// TIA Portal project "Product_Automation_Project" (V17)

(* hardware
DEVICE "S7-1200 station_1"  S7-1200 Station
   slot 0: "Rack_0"  S7-1200 Rack  Rack  V1.0
   slot 1: "PLC_1"  CPU 1214C AC/DC/Rly  6ES7 214-1BG40-0XB0  V4.5
   slot 3: "AQ 1x12BIT_1"  AQ1 signal board  6ES7 232-4HA30-0XB0  V1.0
*)

// ===== PLC "PLC_1"  CPU 1214C AC/DC/Rly =====

VAR_GLOBAL   // PLC tag table "Inputs"
   "PI-100" AT %IW64 : Int;   // Pressure tank sensor
   "H-100.1" AT %I0.1 : Bool;   // System start button
   "H-100.2" AT %I0.2 : Bool;   // System stop button
   "H-100.3" AT %I0.4 : Bool;   // Emergency stop button
   "H-100.4" AT %I0.5 : Bool;   // Emergency reset
   "H-100.5" AT %I0.6 : Bool;   // Pressure tank emptying button
   "Brush_state" AT %I0.0 : Bool;
   "H-100.6" AT %I0.7 : Bool;   // Maintenance reset
END_VAR

VAR_GLOBAL   // PLC tag table "Outputs"
   "PC-100" AT %QW64 : Int;   // Air compressor control
   "OI-100.1" AT %Q0.1 : Bool;   // PID on
   "OI-100.2" AT %Q0.2 : Bool;   // PID off
   "OI-100.3" AT %Q0.3 : Bool;   // Led pressure alarm
   "OI-100.4" AT %Q0.4 : Bool;   // Emergency valve open
   "OI-100.5" AT %Q0.5 : Bool;   // Brush valve closed
   "OI-100.6" AT %Q0.6 : Bool;   // Empty tank indicator
   "OI-100.7" AT %Q0.7 : Bool;
END_VAR

VAR_GLOBAL   // PLC tag table "Variables"
   "PI-100.n" AT %MD0 : Real;   // normalized PI-100 value
   "PI-100.r" AT %MD6 : Real;   // real PI-100 value
   "PC-100.r" AT %MD1 : Real;   // real PC-100 value
   "PC-100.n" AT %MD8 : Real;   // normalized PC-100 value
   "PI-100.r2" AT %MD12 : Real;   // tank pressure
   "System_output" AT %MD16 : Real;   // true system output
   "Brush_pressure" AT %MD20 : Real;   // The ouput pressure of the brush
   "Flip-Flop" AT %M24.0 : Bool;   // Flip-flop
   "Start/Stop value" AT %M24.1 : Bool;
   "Emergency value" AT %M24.2 : Bool;
   "System_state" AT %M24.3 : Bool;
   "Max_pressure_reached" AT %M24.4 : Bool;
   "Emergency_pressure" AT %MD34 : Real;
   "Maintenance_state" AT %M24.5 : Bool;
   "Maintenance_pressure" AT %MD28 : Real;
   "Flip-Flop(1)" AT %M32.0 : Bool;
   "Flip-Flop(2)" AT %M32.1 : Bool;
   "Reset value" AT %M32.2 : Bool;
   "Pressure alarm" AT %M32.4 : Bool;
   "Emergency state" AT %M32.5 : Bool;
   "Brush active/inactive" AT %M32.6 : Bool;
   "min_Output_Reached" AT %M32.7 : Bool;
END_VAR

VAR_GLOBAL   // PLC tag table "Clock_pulses"
   "Clock_Byte(1)" AT %MB150 : Byte;
   "Clock_10Hz(1)" AT %M150.0 : Bool;
   "Clock_5Hz(1)" AT %M150.1 : Bool;
   "Clock_2.5Hz(1)" AT %M150.2 : Bool;
   "Clock_2Hz(1)" AT %M150.3 : Bool;
   "Clock_1.25Hz(1)" AT %M150.4 : Bool;
   "Clock_1Hz(1)" AT %M150.5 : Bool;
   "Clock_0.625Hz(1)" AT %M150.6 : Bool;
   "Clock_0.5Hz(1)" AT %M150.7 : Bool;
END_VAR

DATA_BLOCK "Bool->Real_DB"   // DB1
{ S7_Optimized_Access := 'TRUE' }
VERSION : 0.1
// stored: InstanceOfName Bool->Real
"Bool->Real"
BEGIN
END_DATA_BLOCK

DATA_BLOCK "Integrating_process_DB"   // DB4
{ S7_Optimized_Access := 'TRUE' }
VERSION : 2.01
// stored: InstanceOfName LSim_I
"LSim_I"
BEGIN
END_DATA_BLOCK

DATA_BLOCK "System_state_FB_DB"   // DB5
{ S7_Optimized_Access := 'TRUE' }
VERSION : 0.1
// stored: InstanceOfName System_state_FB
"System_state_FB"
BEGIN
END_DATA_BLOCK

DATA_BLOCK "Emergency_valve_open_DB"   // DB6
{ S7_Optimized_Access := 'TRUE' }
VERSION : 0.1
// stored: InstanceOfName Bool->Real
"Bool->Real"
BEGIN
END_DATA_BLOCK

DATA_BLOCK "Maintenance_DB"   // DB7
{ S7_Optimized_Access := 'TRUE' }
VERSION : 0.1
// stored: InstanceOfName Bool->Real
"Bool->Real"
BEGIN
END_DATA_BLOCK

DATA_BLOCK "Leds_Logic_DB"   // DB8
{ S7_Optimized_Access := 'TRUE' }
VERSION : 0.1
// stored: InstanceOfName Leds_Logic
"Leds_Logic"
BEGIN
END_DATA_BLOCK

DATA_BLOCK "Pressure_alarm_DB"   // DB10
{ S7_Optimized_Access := 'TRUE' }
VERSION : 0.1
// stored: InstanceOfName Pressure_alarm
"Pressure_alarm"
BEGIN
END_DATA_BLOCK

FUNCTION_BLOCK "Signal_scaling"   // FB1, LAD
TITLE = Signal scaling
{ S7_Optimized_Access := 'TRUE' }
VERSION : 0.1
// Here we have the process of scaling the input signal of the PID
   VAR_INPUT
      Input_value : Int;
   END_VAR
   VAR_OUTPUT
      Output_value : Real;
   END_VAR
   VAR_IN_OUT
      Normalized_value : Real;
   END_VAR
BEGIN

REGION Network 1: Normalizing input value
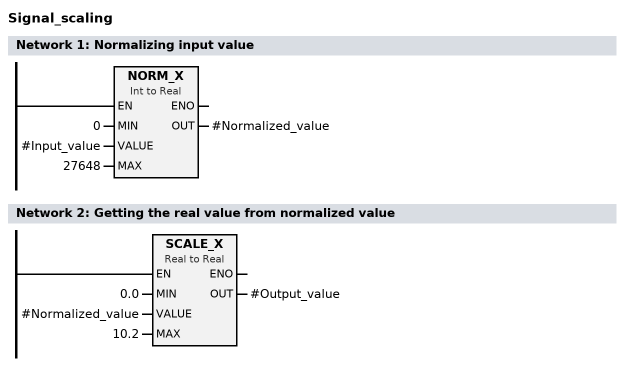
   RUNG wire#powerrail
      { S7_Templates := "[SrcType := Int, DestType := Real]" } Normalize(min := 0, value := #Input_value, max := 27648, out => #Normalized_value)
   END_RUNG
   // the same network as SCL:
   #Normalized_value := NORM_X(MIN := 0, VALUE := #Input_value, MAX := 27648);
END_REGION

REGION Network 2: Getting the real value from normalized value
   RUNG wire#powerrail
      { S7_Templates := "[SrcType := Real, DestType := Real]" } Scale(min := 0.0, value := #Normalized_value, max := 10.2, out => #Output_value)
   END_RUNG
   // the same network as SCL:
   #Output_value := SCALE_X(MIN := 0.0, VALUE := #Normalized_value, MAX := 10.2);
END_REGION
END_FUNCTION_BLOCK

FUNCTION_BLOCK "Bool->Real"   // FB2, SCL
{ S7_Optimized_Access := 'TRUE' }
VERSION : 0.1
   VAR_INPUT
      Boolean_input : Bool;
      Input_pressure : Real;
   END_VAR
   VAR_OUTPUT
      Output_pressure : Real;
   END_VAR
BEGIN
   IF #Boolean_input THEN
       #Output_pressure := #Input_pressure;
   ELSE
       #Output_pressure := 0;
   END_IF;
END_FUNCTION_BLOCK

FUNCTION_BLOCK "System_state_FB"   // FB3, FBD
TITLE = System functioning logic
{ S7_Optimized_Access := 'TRUE' }
VERSION : 0.1
BEGIN

REGION Network 1: System state logic
   // Both Emergency value and Start/Stop value must be "1"
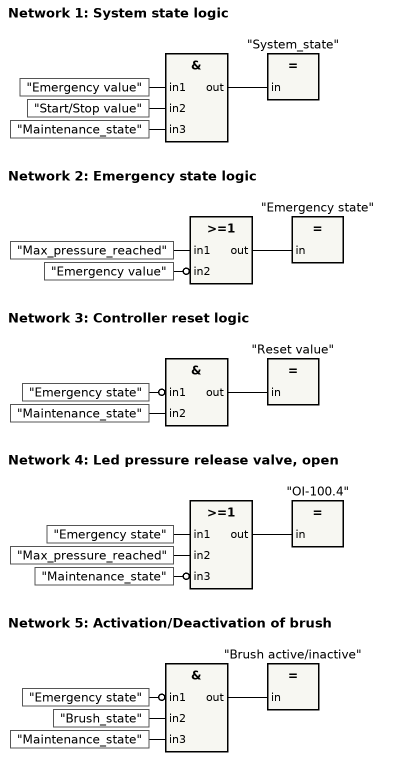
   "System_state" := "Emergency value" AND "Start/Stop value" AND "Maintenance_state";
END_REGION

REGION Network 2: Emergency state logic
   // if max pressure (10.5) is reached or emergency value is 1 than the emergency state is "1"
   "Emergency state" := "Max_pressure_reached" OR NOT "Emergency value";
END_REGION

REGION Network 3: Controller reset logic
   // If both are not pressed then Reset value is 1 -> 0 in controller
   "Reset value" := NOT "Emergency state" AND "Maintenance_state";
END_REGION

REGION Network 4: Led pressure release valve, open
   "OI-100.4" := "Emergency state" OR "Max_pressure_reached" OR NOT "Maintenance_state";
END_REGION

REGION Network 5: Activation/Deactivation of brush
   // Emergency state is active when 0 and inactive when 1
   "Brush active/inactive" := NOT "Emergency state" AND "Brush_state" AND "Maintenance_state";
END_REGION
END_FUNCTION_BLOCK

FUNCTION_BLOCK "Leds_Logic"   // FB4, SCL
{ S7_Optimized_Access := 'TRUE' }
VERSION : 0.1
   VAR_INPUT
      Input : Bool;
   END_VAR
   VAR_OUTPUT
      Output1 : Bool;
      Output2 : Bool;
   END_VAR
BEGIN
   IF #Input THEN
       #Output1 := 1;
       #Output2 := 0;
   ELSE
       #Output2 := 1;
       #Output1 := 0;
   END_IF;
END_FUNCTION_BLOCK

FUNCTION_BLOCK "Pressure_alarm"   // FB5, SCL
{ S7_Optimized_Access := 'TRUE' }
VERSION : 0.1
   VAR_INPUT
      Input : Real;
   END_VAR
   VAR_OUTPUT
      Output : Bool;
   END_VAR
BEGIN
   IF #Input>=10.2 AND #Input<10.5 THEN
       #Output := 1;
   ELSE
       #Output := 0;
   END_IF;
END_FUNCTION_BLOCK

FUNCTION_BLOCK "LSim_I"   // FB56, SCL
{ S7_Optimized_Access := 'TRUE' }
VERSION : 2.01
   VAR_INPUT
      calcParam : Bool;   // recalculate with new parameters
      input : Real;   // input signal
      tmLag1 : Real := 1.0;   // time constant T1 [sec]
      cycle : Real := 0.1;   // cyclic time [sec]
      maxOut : Real := 100.0;   // max. output limit
      minOut : Real;   // min. output limit
      reset : Bool;   // resets all relevant parameters to ‘0’ including the output
   END_VAR
   VAR_OUTPUT
      error : Bool;   // error (#tmLag1 <= 0)
      status : Word;   // status (if #tmLag1 <= 0 then status = 16#8001)
      maxReached : Bool;   // output has reached max. limit
      minReached : Bool;   // output has reached min. limit
      output : Real;   // output signal (if #error = FALSE)
   END_VAR
   VAR
      statRxn1 : Real;   // delayed input signal (n-1)
      statRyn1 : Real;   // delayed output signal (n-1)
      statRa1 : Real;
      statRb1 : Real;
      statOverfirst : Bool;
      statOutput : Real;   // output signal
   END_VAR
BEGIN
   //=============================================================================
   //SIEMENS AG
   //(c)Copyright 2017 All Rights Reserved
   //-----------------------------------------------------------------------------
   //Library:       Library for Controlled System Simulation
   //Tested with:   S7-1500 FW V2.0 / S7-1200 FW V4.2
   //Engineering:   STEP 7 V14 Upd2 (TIA Portal)
   //Restrictions:  Cyclic interrupt
   //Requirements:  memory card needed for S7-1500
   //Functionality: Simulation of a I-System
   //
   //             1
   //  F(p) = -----------
   //         (tmLag1*p)
   //          
   //  Call the simulation in a cyclic interrupt with
   //  cyclic interrupt time at least = tmLag1/10!
   //-----------------------------------------------------------------------------
   //Change log table:
   //Version  Date       Expert in charge                Changes applied
   //02.00.00 03.02.2016 Siemens Industry Online Support Release (STEP 7 V13 SP1)
   //02.00.01 02.03.2017 Siemens Industry Online Support Release (STEP 7 V14)
   //=============================================================================

   // check parameter
   IF #tmLag1 <= 0 THEN
     #error := True;
     #status := W#16#8001;     // Parameter Error
     #statRxn1 := 0.0;
     #statRyn1 := 0.0;
     #statOutput := 0;
     #output := 0;
     RETURN;
   ELSE
     #error := FALSE;
     #status := W#16#0000;     // no error
   END_IF;

   // calculates the z-parameter for the difference equatation
   IF #calcParam = True OR NOT #statOverfirst THEN
   #statOverfirst:=1;
     // Calculate z-parameters for IT1-System
   #statRb1 := #cycle/#tmLag1;
   #statRa1 := -1;

   END_IF;

   // reset Memory
   IF #reset = True THEN
     #statRxn1 := 0.0;
     #statRyn1 := 0.0;
     #statOutput:=0;
   END_IF;

   // save delayed output-signals
   #statRyn1:= #statOutput;

   // difference equatation for the I-system
   #statOutput := #statRxn1* #statRb1 - #statRyn1*#statRa1;

   // save delayed input-signals
   #statRxn1 := #input;

   // max limit of acutating variable
   IF #statOutput > #maxOut THEN
     #statOutput := #maxOut;
     #maxReached:= True;
   ELSE
     #maxReached := False;
   END_IF;

   // min limit of acutating variable
   IF #statOutput < #minOut THEN
     #statOutput := #minOut;
     #minReached := True;
   ELSE
     #minReached := False;
   END_IF;

   #output := #statOutput;
END_FUNCTION_BLOCK

ORGANIZATION_BLOCK "Main"   // OB1, LAD, ProgramCycle
TITLE = "Main Program Sweep (Cycle)"
{ S7_Optimized_Access := 'TRUE' }
VERSION : 0.1
   VAR_INPUT
      Initial_Call : Bool;   // Initial call of this OB
      Remanence : Bool;   // =True, if remanent data are available
   END_VAR
BEGIN

REGION Network 1: Start/Stop logic
   // if start button is pressed then Start/Stop value becomes 1 and if emergency value is also 1 then system state is 1
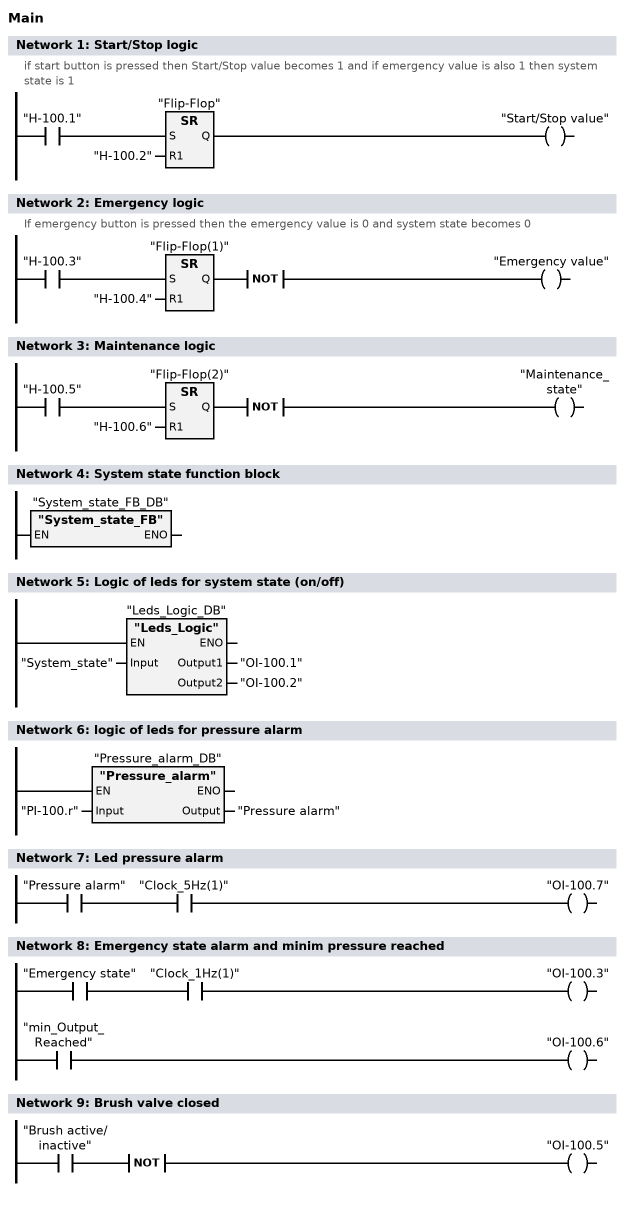
   RUNG wire#powerrail
      Contact( "H-100.1" )
      S_SR(operand := "Flip-Flop", r1 := "H-100.2")
      Coil( "Start/Stop value" )
   END_RUNG
   // the same network as SCL:
   IF "H-100.1" THEN
       "Flip-Flop" := TRUE;   // SR flip-flop
   END_IF;
   IF "H-100.2" THEN "Flip-Flop" := FALSE; END_IF;
   "Start/Stop value" := "Flip-Flop";
END_REGION

REGION Network 2: Emergency logic
   // If emergency button is pressed then the emergency value is 0 and system state becomes 0
   RUNG wire#powerrail
      Contact( "H-100.3" )
      S_SR(operand := "Flip-Flop(1)", r1 := "H-100.4")
      Not()
      Coil( "Emergency value" )
   END_RUNG
   // the same network as SCL:
   IF "H-100.3" THEN
       "Flip-Flop(1)" := TRUE;   // SR flip-flop
   END_IF;
   IF "H-100.4" THEN "Flip-Flop(1)" := FALSE; END_IF;
   "Emergency value" := NOT "Flip-Flop(1)";
END_REGION

REGION Network 3: Maintenance logic
   RUNG wire#powerrail
      Contact( "H-100.5" )
      S_SR(operand := "Flip-Flop(2)", r1 := "H-100.6")
      Not()
      Coil( "Maintenance_state" )
   END_RUNG
   // the same network as SCL:
   IF "H-100.5" THEN
       "Flip-Flop(2)" := TRUE;   // SR flip-flop
   END_IF;
   IF "H-100.6" THEN "Flip-Flop(2)" := FALSE; END_IF;
   "Maintenance_state" := NOT "Flip-Flop(2)";
END_REGION

REGION Network 4: System state function block
   RUNG wire#powerrail
      "System_state_FB_DB"()
   END_RUNG
   // the same network as SCL:
   "System_state_FB_DB"();   // "System_state_FB"
END_REGION

REGION Network 5: Logic of leds for system state (on/off)
   RUNG wire#powerrail
      "Leds_Logic_DB"(Input := "System_state", Output1 => "OI-100.1", Output2 => "OI-100.2")
   END_RUNG
   // the same network as SCL:
   "Leds_Logic_DB"(Input := "System_state", Output1 => "OI-100.1", Output2 => "OI-100.2");   // "Leds_Logic"
END_REGION

REGION Network 6: logic of leds for pressure alarm
   RUNG wire#powerrail
      "Pressure_alarm_DB"(Input := "PI-100.r", Output => "Pressure alarm")
   END_RUNG
   // the same network as SCL:
   "Pressure_alarm_DB"(Input := "PI-100.r", Output => "Pressure alarm");   // "Pressure_alarm"
END_REGION

REGION Network 7: Led pressure alarm
   RUNG wire#powerrail
      Contact( "Pressure alarm" )
      Contact( "Clock_5Hz(1)" )
      Coil( "OI-100.7" )
   END_RUNG
   // the same network as SCL:
   "OI-100.7" := "Pressure alarm" AND "Clock_5Hz(1)";
END_REGION

REGION Network 8: Emergency state alarm and minim pressure reached
   RUNG wire#powerrail
      Contact( "Emergency state" )
      Contact( "Clock_1Hz(1)" )
      Coil( "OI-100.3" )
   END_RUNG
   RUNG wire#powerrail
      Contact( "min_Output_Reached" )
      Coil( "OI-100.6" )
   END_RUNG
   // the same network as SCL:
   "OI-100.3" := "Emergency state" AND "Clock_1Hz(1)";
   "OI-100.6" := "min_Output_Reached";
END_REGION

REGION Network 9: Brush valve closed
   RUNG wire#powerrail
      Contact( "Brush active/inactive" )
      Not()
      Coil( "OI-100.5" )
   END_RUNG
   // the same network as SCL:
   "OI-100.5" := NOT "Brush active/inactive";
END_REGION
END_ORGANIZATION_BLOCK

ORGANIZATION_BLOCK "Cyclic interrupt_1"   // OB30, FBD, CyclicInterrupt
TITLE = Main control loop
{ S7_Optimized_Access := 'TRUE' }
VERSION : 0.1
   VAR_INPUT
      Initial_Call : Bool;   // Initial call of this OB
      Event_Count : Int;   // Events discarded
   END_VAR
BEGIN

REGION Network 1: PID
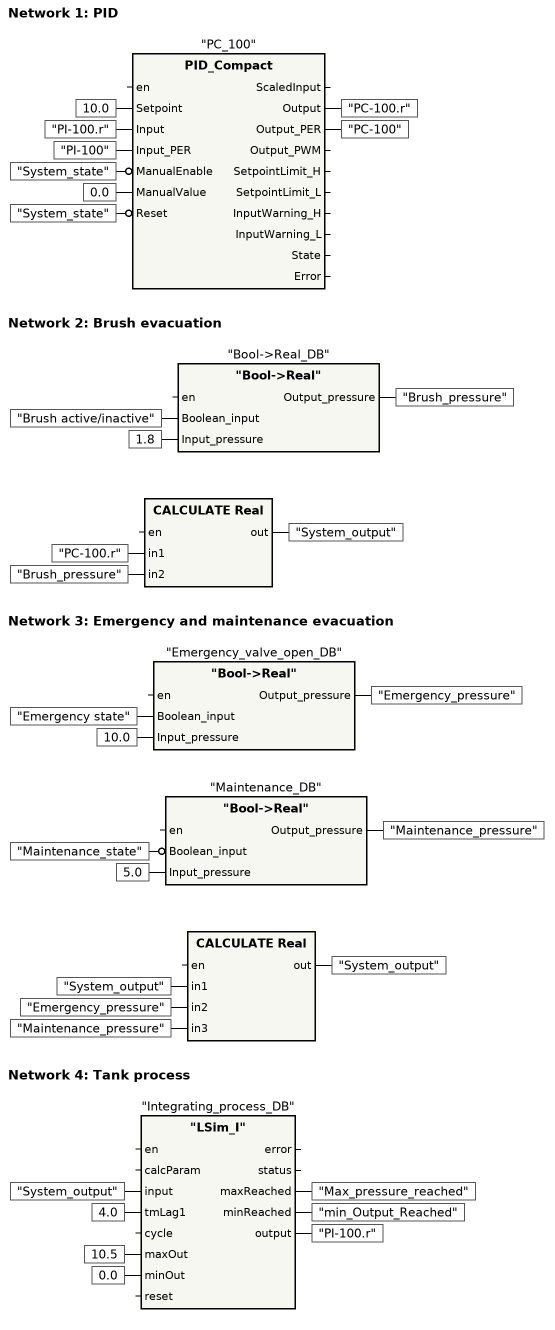
   "PC_100"(Setpoint := 10.0,   // PID_Compact
            Input := "PI-100.r",
            Input_PER := "PI-100",
            ManualEnable := NOT "System_state",
            ManualValue := 0.0,
            Reset := NOT "System_state",
            Output => "PC-100.r",
            Output_PER => "PC-100");
END_REGION

REGION Network 2: Brush evacuation
   "Bool->Real_DB"(Boolean_input := "Brush active/inactive",   // "Bool->Real"
                   Input_pressure := 1.8,
                   Output_pressure => "Brush_pressure");
   "System_output" := "PC-100.r"-"Brush_pressure";
END_REGION

REGION Network 3: Emergency and maintenance evacuation
   "Emergency_valve_open_DB"(Boolean_input := "Emergency state",   // "Bool->Real"
                           Input_pressure := 10.0,
                           Output_pressure => "Emergency_pressure");
   "Maintenance_DB"(Boolean_input := NOT "Maintenance_state",   // "Bool->Real"
                    Input_pressure := 5.0,
                    Output_pressure => "Maintenance_pressure");
   "System_output" := "System_output"- "Emergency_pressure" - "Maintenance_pressure";
END_REGION

REGION Network 4: Tank process
   "Integrating_process_DB"(input := "System_output",   // "LSim_I"
                           tmLag1 := 4.0,
                           maxOut := 10.5,
                           minOut := 0.0,
                           maxReached => "Max_pressure_reached",
                           minReached => "min_Output_Reached",
                           output => "PI-100.r");
END_REGION
END_ORGANIZATION_BLOCK